// TIA Portal V17 export
// export: Created 2024-09-02T12:49:59.6784683Z, ExportSetting WithDefaults, DisplayName Totally Integrated Automation Portal, DisplayVersion V17, DisplayName TIA Portal Openness, DisplayVersion V17, DisplayName TIA Portal Version Control Interface, DisplayVersion V17, DisplayName STEP 7 Professional, DisplayVersion V17, DisplayName STEP 7 Safety, DisplayVersion V17, DisplayName WinCC Professional, DisplayVersion V17
FUNCTION_BLOCK "GraFB_Hand_21_30"   // FB1172, GRAPH
TITLE = GRAPH FB
AUTHOR : OlegFuehrus
FAMILY : SK
NAME : SK
VERSION : 0.1
// Hand functions / Handfunktionen
// stored: AcknowledgeErrorsRequired true, AutoNumber true, ExtensionBlockName LTLL_ManualGraphExt, GraphVersion 4.0, InitialValuesAcquisition false, IsIECCheckEnabled false, LanguageInNetworks LAD, LockOperatingMode false, PermanentILProcessingInMANMode true, SetENOAutomatically false, SkipSteps false, UDAEnableTagReadback false, WithAlarmHandling true
   // inherited from GRAPH_BASE
   VAR
      OFF_SQ_BASE : Bool;
   END_VAR
   VAR_INPUT
      OFF_SQ : Bool;
      INIT_SQ : Bool;
      ACK_EF : Bool;
      S_PREV : Bool;
      S_NEXT : Bool;
      SW_AUTO : Bool;
      SW_TAP : Bool;
      SW_MAN : Bool;
      S_SEL : Int;
      S_ON : Bool;
      S_OFF : Bool;
      T_PUSH : Bool;
   END_VAR
   VAR_OUTPUT
      S_NO : Int;
      S_MORE : Bool;
      S_ACTIVE : Bool;
      ERR_FLT : Bool;
      AUTO_ON : Bool;
      TAP_ON : Bool;
      MAN_ON : Bool;
   END_VAR
   VAR
      extBlock { S7_SetPoint := 'True'} : "LTLL_ManualGraphExt";
   END_VAR
   VAR_TEMP
      t_FrgHand : Bool;   // Freigabe Handbetrieb / Enable manual operation
      t_Service : Bool;   // Servicebetrieb aktiv / Service operation active
   END_VAR
BEGIN
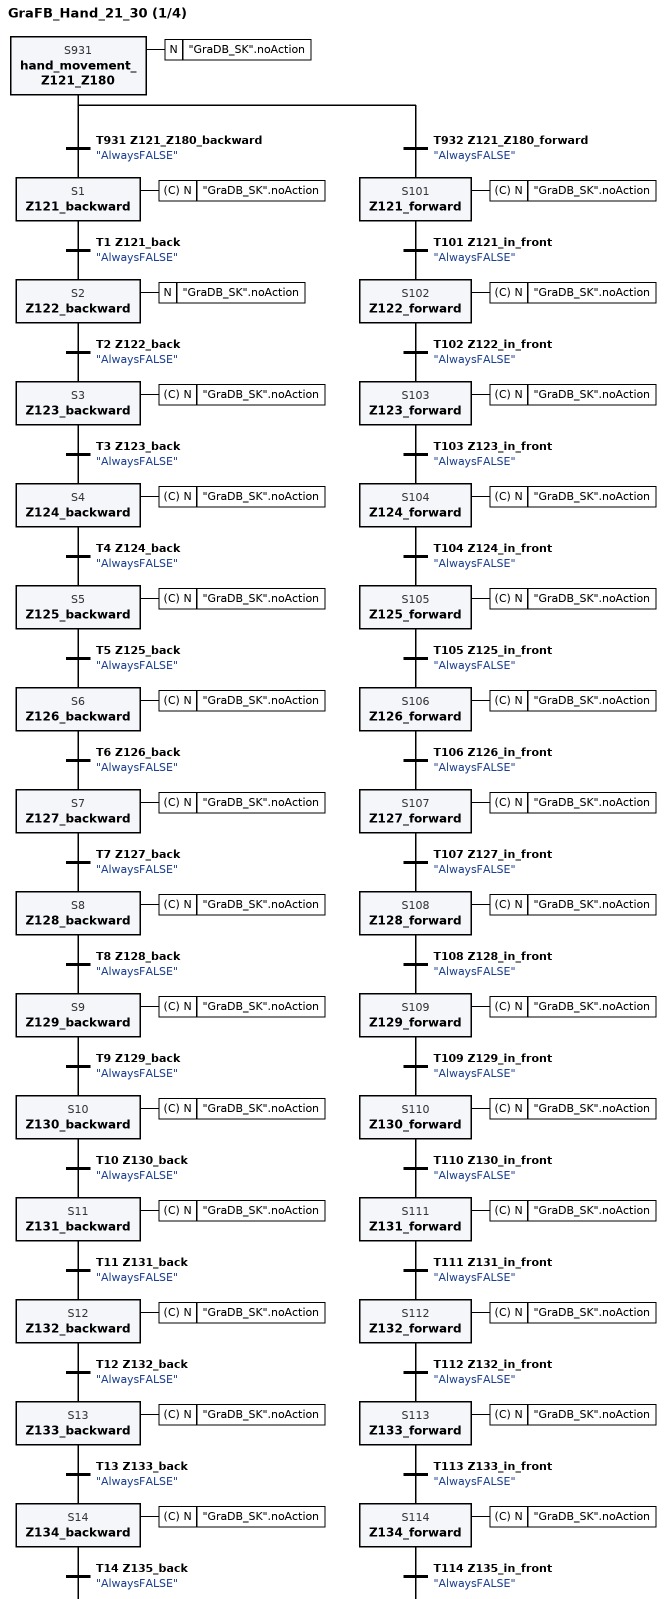
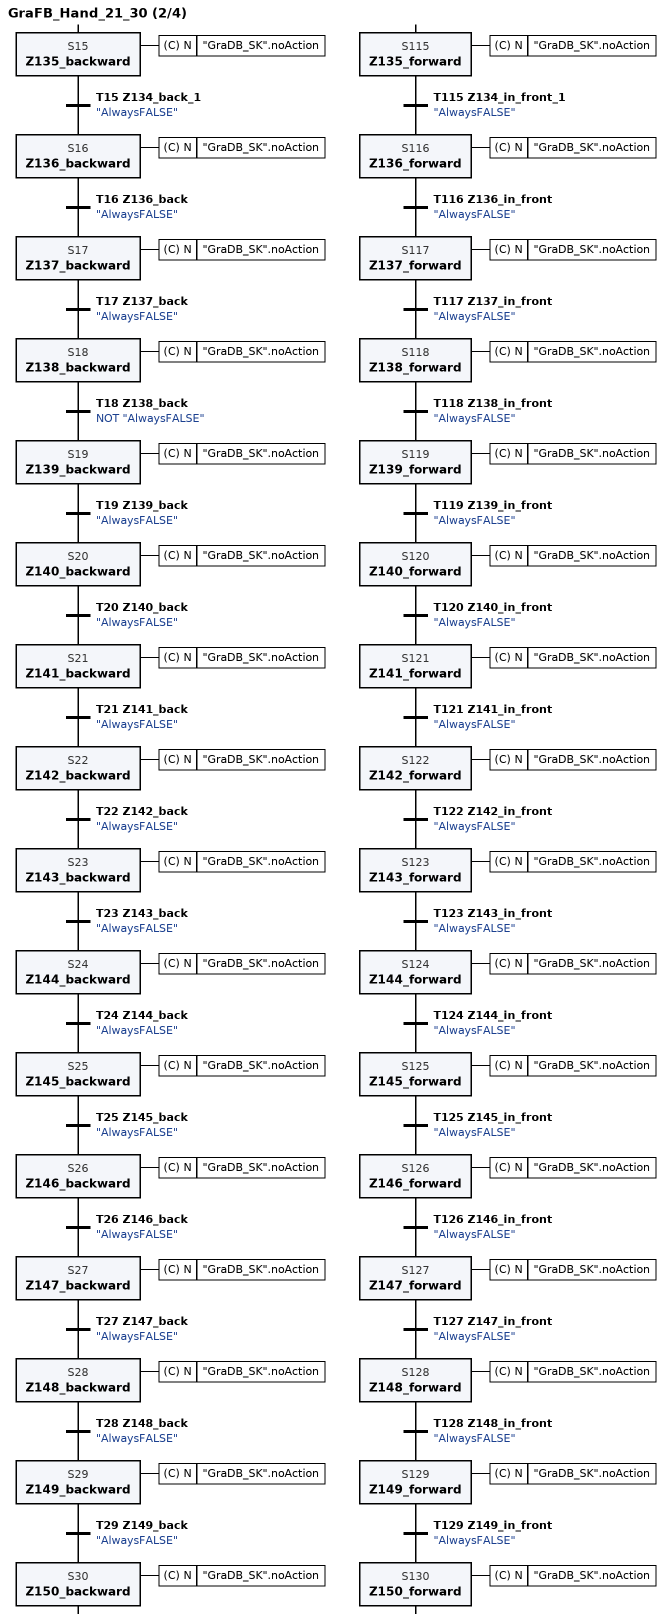
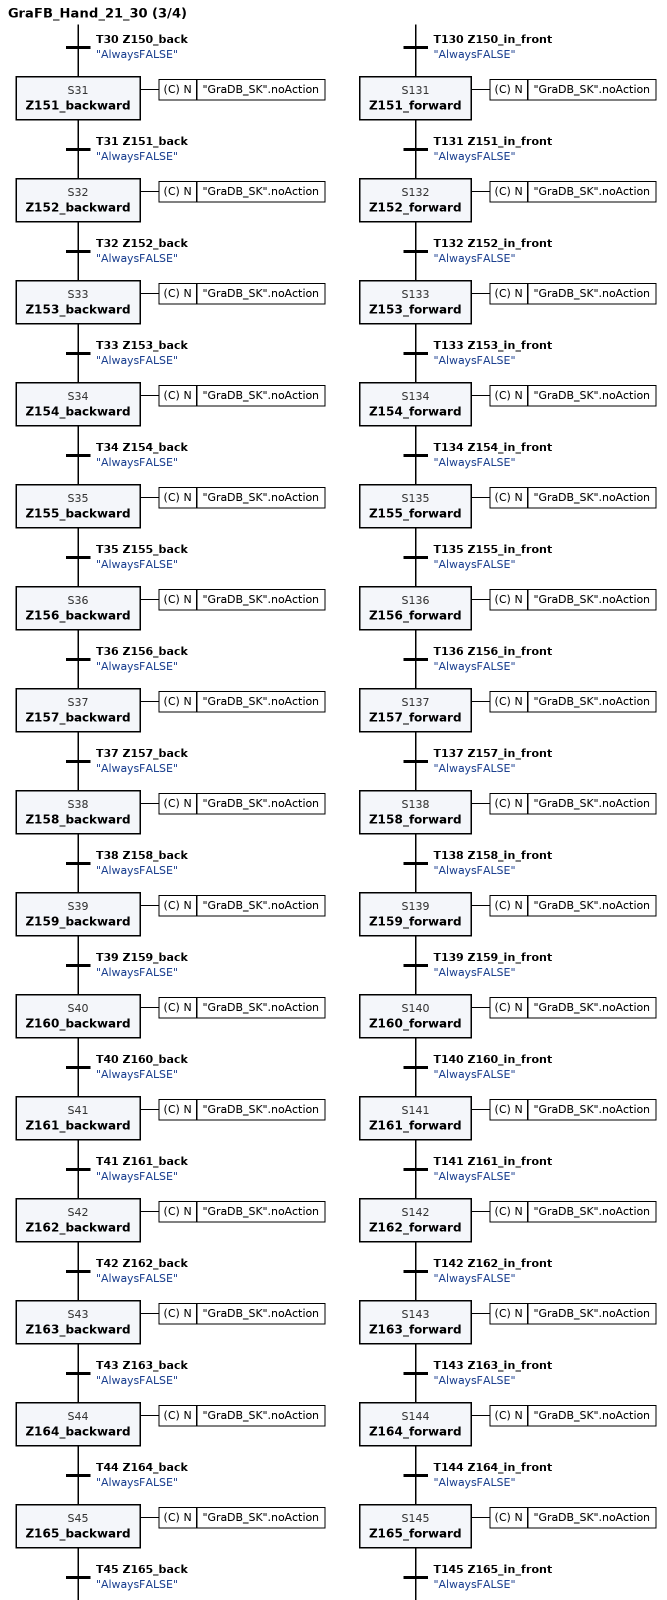
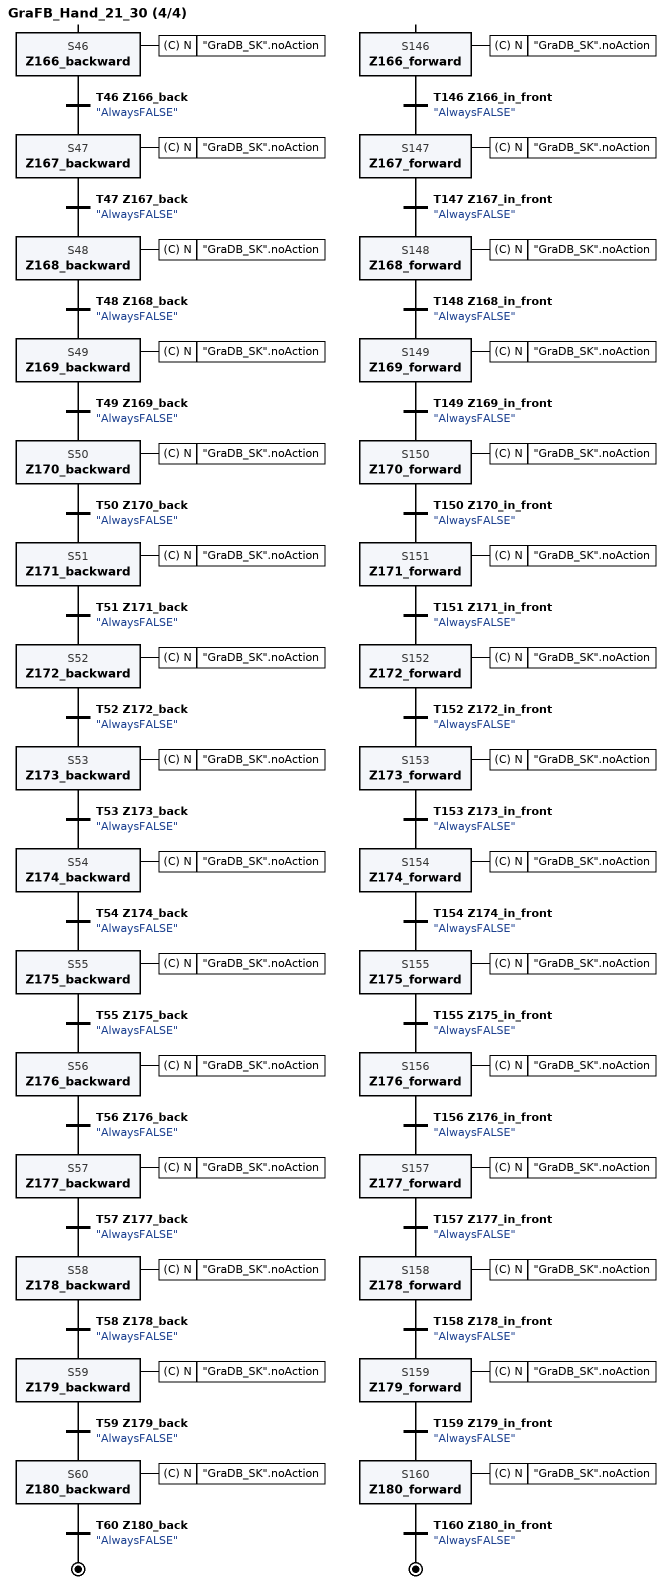
   // permanent pre-instructions
   NETWORK 1
   TITLE = HMI Lite Pass on data / HMI Lite Daten weiterreichen
      #extBlock.input := "LTLL_ManualGraphControl_OP70".screen[0].input;
   NETWORK 2
   TITLE = Instance DB Name query and pass on / Instanz DB Name abfragen und weiterreichen
      GetInstanceName(size := 0, OUT => #extBlock.input.instanceName);
   NETWORK 3
   TITLE = Interlocks Permanent machining, manual Approve and service / Interlocks Permanent Bearbeiten, Handfreigabe und Service
      IF NOT #RT_DATA.MOP.IL_PERM THEN #RT_DATA.MOP.IL_PERM := TRUE; END_IF;
      #t_FrgHand := "AnwDB_OperatingModes_OP70".BA[0]."mode_hand+start";
      #t_Service := "AnwDB_OperatingModes_OP70".BA[0].mode_service;

   // sequencer 1: Sequencer 1
   STEP hand_movement_Z121_Z180:   // S931, max time T#10S, warning time T#7S: Step commentary / Schrittkommentar
      interlock C := (none);   // hand_bereich_Z001_Z005
      supervision V := (none);   // hand_bereich_Z001_Z005
              N    "GraDB_SK".noAction
   END_STEP
   TRANSITION Z121_Z180_backward FROM hand_movement_Z121_Z180 TO Z121_backward   // T931
      := "AlwaysFALSE";
   END_TRANSITION
   TRANSITION Z121_Z180_forward FROM hand_movement_Z121_Z180 TO Z121_forward   // T932
      := "AlwaysFALSE";
   END_TRANSITION
   STEP Z121_backward:   // S1, max time T#10S, warning time T#7S
      interlock C := "AlwaysFALSE";   // Z121_zur
      supervision V := NOT #Z121_back.TT AND (#Z121_backward.T > T#5S);   // Z121_zur
      (C)     N    "GraDB_SK".noAction
   END_STEP
   TRANSITION Z121_back FROM Z121_backward TO Z122_backward   // T1
      := "AlwaysFALSE";
   END_TRANSITION
   STEP Z122_backward:   // S2, max time T#10S, warning time T#7S
      interlock C := "AlwaysFALSE";   // Z122_zur
      supervision V := NOT #Z122_back.TT AND (#Z122_backward.T > T#5S);   // Z122_zur
              N    "GraDB_SK".noAction
   END_STEP
   TRANSITION Z122_back FROM Z122_backward TO Z123_backward   // T2
      := "AlwaysFALSE";
   END_TRANSITION
   STEP Z123_backward:   // S3, max time T#10S, warning time T#7S
      interlock C := "AlwaysFALSE";   // Z123_zur
      supervision V := NOT #Z123_back.TT AND (#Z123_backward.T > T#5S);   // Z123_zur
      (C)     N    "GraDB_SK".noAction
   END_STEP
   TRANSITION Z123_back FROM Z123_backward TO Z124_backward   // T3
      := "AlwaysFALSE";
   END_TRANSITION
   STEP Z124_backward:   // S4, max time T#10S, warning time T#7S
      interlock C := "AlwaysFALSE";   // Z124_zur
      supervision V := NOT #Z124_back.TT AND (#Z124_backward.T > T#5S);   // Z124_zur
      (C)     N    "GraDB_SK".noAction
   END_STEP
   TRANSITION Z124_back FROM Z124_backward TO Z125_backward   // T4
      := "AlwaysFALSE";
   END_TRANSITION
   STEP Z125_backward:   // S5, max time T#10S, warning time T#7S
      interlock C := "AlwaysFALSE";   // Z125_zur
      supervision V := NOT #Z125_back.TT AND (#Z125_backward.T > T#5S);   // Z125_zur
      (C)     N    "GraDB_SK".noAction
   END_STEP
   TRANSITION Z125_back FROM Z125_backward TO Z126_backward   // T5
      := "AlwaysFALSE";
   END_TRANSITION
   STEP Z121_forward:   // S101, max time T#10S, warning time T#7S
      interlock C := "AlwaysFALSE";   // Z121_vor
      supervision V := NOT #Z121_in_front.TT AND (#Z121_forward.T > T#5S);   // Z121_vor
      (C)     N    "GraDB_SK".noAction
   END_STEP
   TRANSITION Z121_in_front FROM Z121_forward TO Z122_forward   // T101
      := "AlwaysFALSE";
   END_TRANSITION
   STEP Z122_forward:   // S102, max time T#10S, warning time T#7S
      interlock C := "AlwaysFALSE";   // Z122_vor
      supervision V := NOT #Z122_in_front.TT AND (#Z122_forward.T > T#5S);   // Z122_vor
      (C)     N    "GraDB_SK".noAction
   END_STEP
   TRANSITION Z122_in_front FROM Z122_forward TO Z123_forward   // T102
      := "AlwaysFALSE";
   END_TRANSITION
   STEP Z123_forward:   // S103, max time T#10S, warning time T#7S
      interlock C := "AlwaysFALSE";   // Z123_vor
      supervision V := NOT #Z123_in_front.TT AND (#Z123_forward.T > T#5S);   // Z123_vor
      (C)     N    "GraDB_SK".noAction
   END_STEP
   TRANSITION Z123_in_front FROM Z123_forward TO Z124_forward   // T103
      := "AlwaysFALSE";
   END_TRANSITION
   STEP Z124_forward:   // S104, max time T#10S, warning time T#7S
      interlock C := "AlwaysFALSE";   // Z124_vor
      supervision V := NOT #Z124_in_front.TT AND (#Z124_forward.T > T#5S);   // Z124_vor
      (C)     N    "GraDB_SK".noAction
   END_STEP
   TRANSITION Z124_in_front FROM Z124_forward TO Z125_forward   // T104
      := "AlwaysFALSE";
   END_TRANSITION
   STEP Z125_forward:   // S105, max time T#10S, warning time T#7S
      interlock C := "AlwaysFALSE";   // Z125_vor
      supervision V := NOT #Z125_in_front.TT AND (#Z125_forward.T > T#20S);   // Z125_vor
      (C)     N    "GraDB_SK".noAction
   END_STEP
   TRANSITION Z125_in_front FROM Z125_forward TO Z126_forward   // T105
      := "AlwaysFALSE";
   END_TRANSITION
   STEP Z126_backward:   // S6, max time T#10S, warning time T#7S: Cross transport 2 / Quertransport 2
      interlock C := "AlwaysFALSE";   // Z126_zur
      supervision V := NOT #Z126_back.TT AND (#Z126_backward.T > T#5S);   // Z126_zur
      (C)     N    "GraDB_SK".noAction
   END_STEP
   TRANSITION Z126_back FROM Z126_backward TO Z127_backward   // T6
      := "AlwaysFALSE";
   END_TRANSITION
   STEP Z127_backward:   // S7, max time T#10S, warning time T#7S
      interlock C := "AlwaysFALSE";   // Z127_zur
      supervision V := NOT #Z127_back.TT AND (#Z127_backward.T > T#5S);   // Z127_zur
      (C)     N    "GraDB_SK".noAction
   END_STEP
   TRANSITION Z127_back FROM Z127_backward TO Z128_backward   // T7
      := "AlwaysFALSE";
   END_TRANSITION
   STEP Z128_backward:   // S8, max time T#10S, warning time T#7S
      interlock C := "AlwaysFALSE";   // Z128_zur
      supervision V := NOT #Z128_back.TT AND (#Z128_backward.T > T#5S);   // Z128_zur
      (C)     N    "GraDB_SK".noAction
   END_STEP
   TRANSITION Z128_back FROM Z128_backward TO Z129_backward   // T8
      := "AlwaysFALSE";
   END_TRANSITION
   STEP Z129_backward:   // S9, max time T#10S, warning time T#7S
      interlock C := "AlwaysFALSE";   // Z129_zur
      supervision V := NOT #Z129_back.TT AND (#Z129_backward.T > T#5S);   // Z129_zur
      (C)     N    "GraDB_SK".noAction
   END_STEP
   TRANSITION Z129_back FROM Z129_backward TO Z130_backward   // T9
      := "AlwaysFALSE";
   END_TRANSITION
   STEP Z130_backward:   // S10, max time T#10S, warning time T#7S
      interlock C := "AlwaysFALSE";   // Z130_zur
      supervision V := NOT #Z130_back.TT AND (#Z130_backward.T > T#5S);   // Z130_zur
      (C)     N    "GraDB_SK".noAction
   END_STEP
   TRANSITION Z130_back FROM Z130_backward TO Z131_backward   // T10
      := "AlwaysFALSE";
   END_TRANSITION
   STEP Z126_forward:   // S106, max time T#10S, warning time T#7S
      interlock C := "AlwaysFALSE";   // Z126_vor
      supervision V := NOT #Z126_in_front.TT AND (#Z126_forward.T > T#5S);   // Z126_vor
      (C)     N    "GraDB_SK".noAction
   END_STEP
   TRANSITION Z126_in_front FROM Z126_forward TO Z127_forward   // T106
      := "AlwaysFALSE";
   END_TRANSITION
   STEP Z127_forward:   // S107, max time T#10S, warning time T#7S
      interlock C := "AlwaysFALSE";   // Z127_vor
      supervision V := NOT #Z127_in_front.TT AND (#Z127_forward.T > T#5S);   // Z127_vor
      (C)     N    "GraDB_SK".noAction
   END_STEP
   TRANSITION Z127_in_front FROM Z127_forward TO Z128_forward   // T107
      := "AlwaysFALSE";
   END_TRANSITION
   STEP Z128_forward:   // S108, max time T#10S, warning time T#7S
      interlock C := "AlwaysFALSE";   // Z128_vor
      supervision V := NOT #Z128_in_front.TT AND (#Z128_forward.T > T#5S);   // Z128_vor
      (C)     N    "GraDB_SK".noAction
   END_STEP
   TRANSITION Z128_in_front FROM Z128_forward TO Z129_forward   // T108
      := "AlwaysFALSE";
   END_TRANSITION
   STEP Z129_forward:   // S109, max time T#10S, warning time T#7S
      interlock C := "AlwaysFALSE";   // Z129_vor
      supervision V := NOT #Z129_in_front.TT AND (#Z129_forward.T > T#5S);   // Z129_vor
      (C)     N    "GraDB_SK".noAction
   END_STEP
   TRANSITION Z129_in_front FROM Z129_forward TO Z130_forward   // T109
      := "AlwaysFALSE";
   END_TRANSITION
   STEP Z130_forward:   // S110, max time T#10S, warning time T#7S
      interlock C := "AlwaysFALSE";   // Z130_vor
      supervision V := NOT #Z130_in_front.TT AND (#Z130_forward.T > T#5S);   // Z130_vor
      (C)     N    "GraDB_SK".noAction
   END_STEP
   TRANSITION Z130_in_front FROM Z130_forward TO Z131_forward   // T110
      := "AlwaysFALSE";
   END_TRANSITION
   STEP Z131_backward:   // S11, max time T#10S, warning time T#7S
      interlock C := "AlwaysFALSE";   // Z131_zur
      supervision V := NOT #Z131_back.TT AND (#Z131_backward.T > T#5S);   // Z131_zur
      (C)     N    "GraDB_SK".noAction
   END_STEP
   TRANSITION Z131_back FROM Z131_backward TO Z132_backward   // T11
      := "AlwaysFALSE";
   END_TRANSITION
   STEP Z132_backward:   // S12, max time T#10S, warning time T#7S
      interlock C := "AlwaysFALSE";   // Z132_zur
      supervision V := NOT #Z132_back.TT AND (#Z132_backward.T > T#5S);   // Z132_zur
      (C)     N    "GraDB_SK".noAction
   END_STEP
   TRANSITION Z132_back FROM Z132_backward TO Z133_backward   // T12
      := "AlwaysFALSE";
   END_TRANSITION
   STEP Z133_backward:   // S13, max time T#10S, warning time T#7S
      interlock C := "AlwaysFALSE";   // Z133_zur
      supervision V := NOT #Z133_back.TT AND (#Z133_backward.T > T#5S);   // Z133_zur
      (C)     N    "GraDB_SK".noAction
   END_STEP
   TRANSITION Z133_back FROM Z133_backward TO Z134_backward   // T13
      := "AlwaysFALSE";
   END_TRANSITION
   STEP Z134_backward:   // S14, max time T#10S, warning time T#7S
      interlock C := "AlwaysFALSE";   // Z135_zur
      supervision V := NOT #Z135_back.TT AND (#Z134_backward.T > T#5S);   // Z135_zur
      (C)     N    "GraDB_SK".noAction
   END_STEP
   TRANSITION Z135_back FROM Z134_backward TO Z135_backward   // T14
      := "AlwaysFALSE";
   END_TRANSITION
   STEP Z135_backward:   // S15, max time T#10S, warning time T#7S
      interlock C := "AlwaysFALSE";   // Z134_zur
      supervision V := NOT #Z136_back.TT AND (#Z135_backward.T > T#5S);   // Z134_zur
      (C)     N    "GraDB_SK".noAction
   END_STEP
   TRANSITION Z134_back_1 FROM Z135_backward TO Z136_backward   // T15
      := "AlwaysFALSE";
   END_TRANSITION
   STEP Z131_forward:   // S111, max time T#10S, warning time T#7S
      interlock C := "AlwaysFALSE";   // Z131_vor
      supervision V := NOT #Z131_in_front.TT AND (#Z131_forward.T > T#5S);   // Z131_vor
      (C)     N    "GraDB_SK".noAction
   END_STEP
   TRANSITION Z131_in_front FROM Z131_forward TO Z132_forward   // T111
      := "AlwaysFALSE";
   END_TRANSITION
   STEP Z132_forward:   // S112, max time T#10S, warning time T#7S
      interlock C := "AlwaysFALSE";   // Z132_vor
      supervision V := NOT #Z132_in_front.TT AND (#Z132_forward.T > T#5S);   // Z132_vor
      (C)     N    "GraDB_SK".noAction
   END_STEP
   TRANSITION Z132_in_front FROM Z132_forward TO Z133_forward   // T112
      := "AlwaysFALSE";
   END_TRANSITION
   STEP Z133_forward:   // S113, max time T#10S, warning time T#7S
      interlock C := "AlwaysFALSE";   // Z133_vor
      supervision V := NOT #Z133_in_front.TT AND (#Z133_forward.T > T#5S);   // Z133_vor
      (C)     N    "GraDB_SK".noAction
   END_STEP
   TRANSITION Z133_in_front FROM Z133_forward TO Z134_forward   // T113
      := "AlwaysFALSE";
   END_TRANSITION
   STEP Z134_forward:   // S114, max time T#10S, warning time T#7S
      interlock C := "AlwaysFALSE";   // Z135_vor
      supervision V := NOT #Z135_in_front.TT AND (#Z134_forward.T > T#5S);   // Z135_vor
      (C)     N    "GraDB_SK".noAction
   END_STEP
   TRANSITION Z135_in_front FROM Z134_forward TO Z135_forward   // T114
      := "AlwaysFALSE";
   END_TRANSITION
   STEP Z135_forward:   // S115, max time T#10S, warning time T#7S
      interlock C := "AlwaysFALSE";   // Z134_vor
      supervision V := NOT #Z136_in_front.TT AND (#Z135_forward.T > T#5S);   // Z134_vor
      (C)     N    "GraDB_SK".noAction
   END_STEP
   TRANSITION Z134_in_front_1 FROM Z135_forward TO Z136_forward   // T115
      := "AlwaysFALSE";
   END_TRANSITION
   STEP Z136_backward:   // S16, max time T#10S, warning time T#7S
      interlock C := "AlwaysFALSE";   // Z136_zur
      supervision V := NOT #Z136_back.TT AND (#Z136_backward.T > T#5S);   // Z136_zur
      (C)     N    "GraDB_SK".noAction
   END_STEP
   TRANSITION Z136_back FROM Z136_backward TO Z137_backward   // T16
      := "AlwaysFALSE";
   END_TRANSITION
   STEP Z137_backward:   // S17, max time T#10S, warning time T#7S
      interlock C := "AlwaysFALSE";   // Z137_zur
      supervision V := NOT #Z137_back.TT AND (#Z137_backward.T > T#5S);   // Z137_zur
      (C)     N    "GraDB_SK".noAction
   END_STEP
   TRANSITION Z137_back FROM Z137_backward TO Z138_backward   // T17
      := "AlwaysFALSE";
   END_TRANSITION
   STEP Z138_backward:   // S18, max time T#10S, warning time T#7S
      interlock C := "AlwaysFALSE";   // Z138_zur
      supervision V := NOT #Z138_back.TT AND (#Z138_backward.T > T#5S);   // Z138_zur
      (C)     N    "GraDB_SK".noAction
   END_STEP
   TRANSITION Z138_back FROM Z138_backward TO Z139_backward   // T18
      := NOT "AlwaysFALSE";
   END_TRANSITION
   STEP Z139_backward:   // S19, max time T#10S, warning time T#7S
      interlock C := "AlwaysFALSE";   // Z139_zur
      supervision V := NOT #Z139_back.TT AND (#Z139_backward.T > T#5S);   // Z139_zur
      (C)     N    "GraDB_SK".noAction
   END_STEP
   TRANSITION Z139_back FROM Z139_backward TO Z140_backward   // T19
      := "AlwaysFALSE";
   END_TRANSITION
   STEP Z140_backward:   // S20, max time T#10S, warning time T#7S
      interlock C := "AlwaysFALSE";   // Z140_zur
      supervision V := NOT #Z140_back.TT AND (#Z140_backward.T > T#5S);   // Z140_zur
      (C)     N    "GraDB_SK".noAction
   END_STEP
   TRANSITION Z140_back FROM Z140_backward TO Z141_backward   // T20
      := "AlwaysFALSE";
   END_TRANSITION
   STEP Z136_forward:   // S116, max time T#10S, warning time T#7S
      interlock C := "AlwaysFALSE";   // Z136_vor
      supervision V := NOT #Z136_in_front.TT AND (#Z136_forward.T > T#5S);   // Z136_vor
      (C)     N    "GraDB_SK".noAction
   END_STEP
   TRANSITION Z136_in_front FROM Z136_forward TO Z137_forward   // T116
      := "AlwaysFALSE";
   END_TRANSITION
   STEP Z137_forward:   // S117, max time T#10S, warning time T#7S
      interlock C := "AlwaysFALSE";   // Z137_vor
      supervision V := NOT #Z137_in_front.TT AND (#Z137_forward.T > T#5S);   // Z137_vor
      (C)     N    "GraDB_SK".noAction
   END_STEP
   TRANSITION Z137_in_front FROM Z137_forward TO Z138_forward   // T117
      := "AlwaysFALSE";
   END_TRANSITION
   STEP Z138_forward:   // S118, max time T#10S, warning time T#7S
      interlock C := "AlwaysFALSE";   // Z138_vor
      supervision V := NOT #Z138_in_front.TT AND (#Z138_forward.T > T#5S);   // Z138_vor
      (C)     N    "GraDB_SK".noAction
   END_STEP
   TRANSITION Z138_in_front FROM Z138_forward TO Z139_forward   // T118
      := "AlwaysFALSE";
   END_TRANSITION
   STEP Z139_forward:   // S119, max time T#10S, warning time T#7S
      interlock C := "AlwaysFALSE";   // Z139_vor
      supervision V := NOT #Z139_in_front.TT AND (#Z139_forward.T > T#5S);   // Z139_vor
      (C)     N    "GraDB_SK".noAction
   END_STEP
   TRANSITION Z139_in_front FROM Z139_forward TO Z140_forward   // T119
      := "AlwaysFALSE";
   END_TRANSITION
   STEP Z140_forward:   // S120, max time T#10S, warning time T#7S
      interlock C := "AlwaysFALSE";   // Z140_vor
      supervision V := NOT #Z140_in_front.TT AND (#Z140_forward.T > T#5S);   // Z140_vor
      (C)     N    "GraDB_SK".noAction
   END_STEP
   TRANSITION Z140_in_front FROM Z140_forward TO Z141_forward   // T120
      := "AlwaysFALSE";
   END_TRANSITION
   STEP Z141_backward:   // S21, max time T#10S, warning time T#7S
      interlock C := "AlwaysFALSE";   // Z141_zur
      supervision V := NOT #Z141_back.TT AND (#Z141_backward.T > T#10S);   // Z141_zur
      (C)     N    "GraDB_SK".noAction
   END_STEP
   TRANSITION Z141_back FROM Z141_backward TO Z142_backward   // T21
      := "AlwaysFALSE";
   END_TRANSITION
   STEP Z142_backward:   // S22, max time T#10S, warning time T#7S
      interlock C := "AlwaysFALSE";   // Z142_zur
      supervision V := NOT #Z142_back.TT AND (#Z142_backward.T > T#10S);   // Z142_zur
      (C)     N    "GraDB_SK".noAction
   END_STEP
   TRANSITION Z142_back FROM Z142_backward TO Z143_backward   // T22
      := "AlwaysFALSE";
   END_TRANSITION
   STEP Z143_backward:   // S23, max time T#10S, warning time T#7S
      interlock C := "AlwaysFALSE";   // Z143_zur
      supervision V := NOT #Z143_back.TT AND (#Z143_backward.T > T#10S);   // Z143_zur
      (C)     N    "GraDB_SK".noAction
   END_STEP
   TRANSITION Z143_back FROM Z143_backward TO Z144_backward   // T23
      := "AlwaysFALSE";
   END_TRANSITION
   STEP Z144_backward:   // S24, max time T#10S, warning time T#7S
      interlock C := "AlwaysFALSE";   // Z144_zur
      supervision V := NOT #Z144_back.TT AND (#Z144_backward.T > T#5S);   // Z144_zur
      (C)     N    "GraDB_SK".noAction
   END_STEP
   TRANSITION Z144_back FROM Z144_backward TO Z145_backward   // T24
      := "AlwaysFALSE";
   END_TRANSITION
   STEP Z145_backward:   // S25, max time T#10S, warning time T#7S
      interlock C := "AlwaysFALSE";   // Z145_zur
      supervision V := NOT #Z145_back.TT AND (#Z145_backward.T > T#5S);   // Z145_zur
      (C)     N    "GraDB_SK".noAction
   END_STEP
   TRANSITION Z145_back FROM Z145_backward TO Z146_backward   // T25
      := "AlwaysFALSE";
   END_TRANSITION
   STEP Z141_forward:   // S121, max time T#10S, warning time T#7S
      interlock C := "AlwaysFALSE";   // Z141_vor
      supervision V := NOT #Z141_in_front.TT AND (#Z141_forward.T > T#5S);   // Z141_vor
      (C)     N    "GraDB_SK".noAction
   END_STEP
   TRANSITION Z141_in_front FROM Z141_forward TO Z142_forward   // T121
      := "AlwaysFALSE";
   END_TRANSITION
   STEP Z142_forward:   // S122, max time T#10S, warning time T#7S
      interlock C := "AlwaysFALSE";   // Z142_vor
      supervision V := NOT #Z142_in_front.TT AND (#Z142_forward.T > T#10S);   // Z142_vor
      (C)     N    "GraDB_SK".noAction
   END_STEP
   TRANSITION Z142_in_front FROM Z142_forward TO Z143_forward   // T122
      := "AlwaysFALSE";
   END_TRANSITION
   STEP Z143_forward:   // S123, max time T#10S, warning time T#7S
      interlock C := "AlwaysFALSE";   // Z143_vor
      supervision V := NOT #Z143_in_front.TT AND (#Z143_forward.T > T#10S);   // Z143_vor
      (C)     N    "GraDB_SK".noAction
   END_STEP
   TRANSITION Z143_in_front FROM Z143_forward TO Z144_forward   // T123
      := "AlwaysFALSE";
   END_TRANSITION
   STEP Z144_forward:   // S124, max time T#10S, warning time T#7S
      interlock C := "AlwaysFALSE";   // Z144_vor
      supervision V := NOT #Z144_in_front.TT AND (#Z144_forward.T > T#5S);   // Z144_vor
      (C)     N    "GraDB_SK".noAction
   END_STEP
   TRANSITION Z144_in_front FROM Z144_forward TO Z145_forward   // T124
      := "AlwaysFALSE";
   END_TRANSITION
   STEP Z145_forward:   // S125, max time T#10S, warning time T#7S
      interlock C := "AlwaysFALSE";   // Z145_vor
      supervision V := NOT #Z145_in_front.TT AND (#Z145_forward.T > T#5S);   // Z145_vor
      (C)     N    "GraDB_SK".noAction
   END_STEP
   TRANSITION Z145_in_front FROM Z145_forward TO Z146_forward   // T125
      := "AlwaysFALSE";
   END_TRANSITION
   STEP Z146_backward:   // S26, max time T#10S, warning time T#7S
      interlock C := "AlwaysFALSE";   // Z146_zur
      supervision V := NOT #Z146_back.TT AND (#Z146_backward.T > T#5S);   // Z146_zur
      (C)     N    "GraDB_SK".noAction
   END_STEP
   TRANSITION Z146_back FROM Z146_backward TO Z147_backward   // T26
      := "AlwaysFALSE";
   END_TRANSITION
   STEP Z147_backward:   // S27, max time T#10S, warning time T#7S
      interlock C := "AlwaysFALSE";   // Z147_zur
      supervision V := NOT #Z147_back.TT AND (#Z147_backward.T > T#5S);   // Z147_zur
      (C)     N    "GraDB_SK".noAction
   END_STEP
   TRANSITION Z147_back FROM Z147_backward TO Z148_backward   // T27
      := "AlwaysFALSE";
   END_TRANSITION
   STEP Z148_backward:   // S28, max time T#10S, warning time T#7S
      interlock C := "AlwaysFALSE";   // Z148_zur
      supervision V := NOT #Z148_back.TT AND (#Z148_backward.T > T#5S);   // Z148_zur
      (C)     N    "GraDB_SK".noAction
   END_STEP
   TRANSITION Z148_back FROM Z148_backward TO Z149_backward   // T28
      := "AlwaysFALSE";
   END_TRANSITION
   STEP Z149_backward:   // S29, max time T#10S, warning time T#7S
      interlock C := "AlwaysFALSE";   // Z149_zur
      supervision V := NOT #Z149_back.TT AND (#Z149_backward.T > T#5S);   // Z149_zur
      (C)     N    "GraDB_SK".noAction
   END_STEP
   TRANSITION Z149_back FROM Z149_backward TO Z150_backward   // T29
      := "AlwaysFALSE";
   END_TRANSITION
   STEP Z150_backward:   // S30, max time T#10S, warning time T#7S
      interlock C := "AlwaysFALSE";   // Z150_zur
      supervision V := NOT #Z150_back.TT AND (#Z150_backward.T > T#5S);   // Z150_zur
      (C)     N    "GraDB_SK".noAction
   END_STEP
   TRANSITION Z150_back FROM Z150_backward TO Z151_backward   // T30
      := "AlwaysFALSE";
   END_TRANSITION
   STEP Z146_forward:   // S126, max time T#10S, warning time T#7S
      interlock C := "AlwaysFALSE";   // Z146_vor
      supervision V := NOT #Z146_in_front.TT AND (#Z146_forward.T > T#5S);   // Z146_vor
      (C)     N    "GraDB_SK".noAction
   END_STEP
   TRANSITION Z146_in_front FROM Z146_forward TO Z147_forward   // T126
      := "AlwaysFALSE";
   END_TRANSITION
   STEP Z147_forward:   // S127, max time T#10S, warning time T#7S
      interlock C := "AlwaysFALSE";   // Z147_vor
      supervision V := NOT #Z147_in_front.TT AND (#Z147_forward.T > T#5S);   // Z147_vor
      (C)     N    "GraDB_SK".noAction
   END_STEP
   TRANSITION Z147_in_front FROM Z147_forward TO Z148_forward   // T127
      := "AlwaysFALSE";
   END_TRANSITION
   STEP Z148_forward:   // S128, max time T#10S, warning time T#7S
      interlock C := "AlwaysFALSE";   // Z148_vor
      supervision V := NOT #Z148_in_front.TT AND (#Z148_forward.T > T#5S);   // Z148_vor
      (C)     N    "GraDB_SK".noAction
   END_STEP
   TRANSITION Z148_in_front FROM Z148_forward TO Z149_forward   // T128
      := "AlwaysFALSE";
   END_TRANSITION
   STEP Z149_forward:   // S129, max time T#10S, warning time T#7S
      interlock C := "AlwaysFALSE";   // Z149_vor
      supervision V := NOT #Z149_in_front.TT AND (#Z149_forward.T > T#5S);   // Z149_vor
      (C)     N    "GraDB_SK".noAction
   END_STEP
   TRANSITION Z149_in_front FROM Z149_forward TO Z150_forward   // T129
      := "AlwaysFALSE";
   END_TRANSITION
   STEP Z150_forward:   // S130, max time T#10S, warning time T#7S
      interlock C := "AlwaysFALSE";   // Z150_vor
      supervision V := NOT #Z150_in_front.TT AND (#Z150_forward.T > T#5S);   // Z150_vor
      (C)     N    "GraDB_SK".noAction
   END_STEP
   TRANSITION Z150_in_front FROM Z150_forward TO Z151_forward   // T130
      := "AlwaysFALSE";
   END_TRANSITION
   STEP Z151_backward:   // S31, max time T#10S, warning time T#7S: Step commentary / Schrittkommentar
      interlock C := "AlwaysFALSE";   // Z151_zur
      supervision V := NOT #Z151_back.TT AND (#Z151_backward.T > T#5S);   // Z151_zur
      (C)     N    "GraDB_SK".noAction
   END_STEP
   TRANSITION Z151_back FROM Z151_backward TO Z152_backward   // T31
      := "AlwaysFALSE";
   END_TRANSITION
   STEP Z152_backward:   // S32, max time T#10S, warning time T#7S: Step commentary / Schrittkommentar
      interlock C := "AlwaysFALSE";   // Z152_zur
      supervision V := NOT #Z152_back.TT AND (#Z152_backward.T > T#5S);   // Z152_zur
      (C)     N    "GraDB_SK".noAction
   END_STEP
   TRANSITION Z152_back FROM Z152_backward TO Z153_backward   // T32
      := "AlwaysFALSE";
   END_TRANSITION
   STEP Z153_backward:   // S33, max time T#10S, warning time T#7S: Step commentary / Schrittkommentar
      interlock C := "AlwaysFALSE";   // Z153_zur
      supervision V := NOT #Z153_back.TT AND (#Z153_backward.T > T#5S);   // Z153_zur
      (C)     N    "GraDB_SK".noAction
   END_STEP
   TRANSITION Z153_back FROM Z153_backward TO Z154_backward   // T33
      := "AlwaysFALSE";
   END_TRANSITION
   STEP Z154_backward:   // S34, max time T#10S, warning time T#7S: Step commentary / Schrittkommentar
      interlock C := "AlwaysFALSE";   // Z154_zur
      supervision V := NOT #Z154_back.TT AND (#Z154_backward.T > T#5S);   // Z154_zur
      (C)     N    "GraDB_SK".noAction
   END_STEP
   TRANSITION Z154_back FROM Z154_backward TO Z155_backward   // T34
      := "AlwaysFALSE";
   END_TRANSITION
   STEP Z155_backward:   // S35, max time T#10S, warning time T#7S: Step commentary / Schrittkommentar
      interlock C := "AlwaysFALSE";   // Z155_zur
      supervision V := NOT #Z155_back.TT AND (#Z155_backward.T > T#5S);   // Z155_zur
      (C)     N    "GraDB_SK".noAction
   END_STEP
   TRANSITION Z155_back FROM Z155_backward TO Z156_backward   // T35
      := "AlwaysFALSE";
   END_TRANSITION
   STEP Z151_forward:   // S131, max time T#10S, warning time T#7S: Step commentary / Schrittkommentar
      interlock C := "AlwaysFALSE";   // Z151_vor
      supervision V := NOT #Z151_in_front.TT AND (#Z151_forward.T > T#5S);   // Z151_vor
      (C)     N    "GraDB_SK".noAction
   END_STEP
   TRANSITION Z151_in_front FROM Z151_forward TO Z152_forward   // T131
      := "AlwaysFALSE";
   END_TRANSITION
   STEP Z152_forward:   // S132, max time T#10S, warning time T#7S: Step commentary / Schrittkommentar
      interlock C := "AlwaysFALSE";   // Z152_vor
      supervision V := NOT #Z152_in_front.TT AND (#Z152_forward.T > T#5S);   // Z152_vor
      (C)     N    "GraDB_SK".noAction
   END_STEP
   TRANSITION Z152_in_front FROM Z152_forward TO Z153_forward   // T132
      := "AlwaysFALSE";
   END_TRANSITION
   STEP Z153_forward:   // S133, max time T#10S, warning time T#7S: Step commentary / Schrittkommentar
      interlock C := "AlwaysFALSE";   // Z153_vor
      supervision V := NOT #Z153_in_front.TT AND (#Z153_forward.T > T#5S);   // Z153_vor
      (C)     N    "GraDB_SK".noAction
   END_STEP
   TRANSITION Z153_in_front FROM Z153_forward TO Z154_forward   // T133
      := "AlwaysFALSE";
   END_TRANSITION
   STEP Z154_forward:   // S134, max time T#10S, warning time T#7S: Step commentary / Schrittkommentar
      interlock C := "AlwaysFALSE";   // Z154_vor
      supervision V := NOT #Z154_in_front.TT AND (#Z154_forward.T > T#5S);   // Z154_vor
      (C)     N    "GraDB_SK".noAction
   END_STEP
   TRANSITION Z154_in_front FROM Z154_forward TO Z155_forward   // T134
      := "AlwaysFALSE";
   END_TRANSITION
   STEP Z155_forward:   // S135, max time T#10S, warning time T#7S: Step commentary / Schrittkommentar
      interlock C := "AlwaysFALSE";   // Z155_vor
      supervision V := NOT #Z155_in_front.TT AND (#Z155_forward.T > T#5S);   // Z155_vor
      (C)     N    "GraDB_SK".noAction
   END_STEP
   TRANSITION Z155_in_front FROM Z155_forward TO Z156_forward   // T135
      := "AlwaysFALSE";
   END_TRANSITION
   STEP Z156_backward:   // S36, max time T#10S, warning time T#7S: Step commentary / Schrittkommentar
      interlock C := "AlwaysFALSE";   // Z156_zur
      supervision V := NOT #Z156_back.TT AND (#Z156_backward.T > T#5S);   // Z156_zur
      (C)     N    "GraDB_SK".noAction
   END_STEP
   TRANSITION Z156_back FROM Z156_backward TO Z157_backward   // T36
      := "AlwaysFALSE";
   END_TRANSITION
   STEP Z157_backward:   // S37, max time T#10S, warning time T#7S: Step commentary / Schrittkommentar
      interlock C := "AlwaysFALSE";   // Z157_zur
      supervision V := NOT #Z157_back.TT AND (#Z157_backward.T > T#5S);   // Z157_zur
      (C)     N    "GraDB_SK".noAction
   END_STEP
   TRANSITION Z157_back FROM Z157_backward TO Z158_backward   // T37
      := "AlwaysFALSE";
   END_TRANSITION
   STEP Z158_backward:   // S38, max time T#10S, warning time T#7S: Step commentary / Schrittkommentar
      interlock C := "AlwaysFALSE";   // Z158_zur
      supervision V := NOT #Z158_back.TT AND (#Z158_backward.T > T#5S);   // Z158_zur
      (C)     N    "GraDB_SK".noAction
   END_STEP
   TRANSITION Z158_back FROM Z158_backward TO Z159_backward   // T38
      := "AlwaysFALSE";
   END_TRANSITION
   STEP Z159_backward:   // S39, max time T#10S, warning time T#7S: Step commentary / Schrittkommentar
      interlock C := "AlwaysFALSE";   // Z159_zur
      supervision V := NOT #Z159_back.TT AND (#Z159_backward.T > T#5S);   // Z159_zur
      (C)     N    "GraDB_SK".noAction
   END_STEP
   TRANSITION Z159_back FROM Z159_backward TO Z160_backward   // T39
      := "AlwaysFALSE";
   END_TRANSITION
   STEP Z160_backward:   // S40, max time T#10S, warning time T#7S: Step commentary / Schrittkommentar
      interlock C := "AlwaysFALSE";   // Z160_zur
      supervision V := NOT #Z160_back.TT AND (#Z160_backward.T > T#5S);   // Z160_zur
      (C)     N    "GraDB_SK".noAction
   END_STEP
   TRANSITION Z160_back FROM Z160_backward TO Z161_backward   // T40
      := "AlwaysFALSE";
   END_TRANSITION
   STEP Z156_forward:   // S136, max time T#10S, warning time T#7S: Step commentary / Schrittkommentar
      interlock C := "AlwaysFALSE";   // Z156_vor
      supervision V := NOT #Z156_in_front.TT AND (#Z156_forward.T > T#5S);   // Z156_vor
      (C)     N    "GraDB_SK".noAction
   END_STEP
   TRANSITION Z156_in_front FROM Z156_forward TO Z157_forward   // T136
      := "AlwaysFALSE";
   END_TRANSITION
   STEP Z157_forward:   // S137, max time T#10S, warning time T#7S: Step commentary / Schrittkommentar
      interlock C := "AlwaysFALSE";   // Z157_vor
      supervision V := NOT #Z157_in_front.TT AND (#Z157_forward.T > T#5S);   // Z157_vor
      (C)     N    "GraDB_SK".noAction
   END_STEP
   TRANSITION Z157_in_front FROM Z157_forward TO Z158_forward   // T137
      := "AlwaysFALSE";
   END_TRANSITION
   STEP Z158_forward:   // S138, max time T#10S, warning time T#7S: Step commentary / Schrittkommentar
      interlock C := "AlwaysFALSE";   // Z158_vor
      supervision V := NOT #Z158_in_front.TT AND (#Z158_forward.T > T#5S);   // Z158_vor
      (C)     N    "GraDB_SK".noAction
   END_STEP
   TRANSITION Z158_in_front FROM Z158_forward TO Z159_forward   // T138
      := "AlwaysFALSE";
   END_TRANSITION
   STEP Z159_forward:   // S139, max time T#10S, warning time T#7S: Step commentary / Schrittkommentar
      interlock C := "AlwaysFALSE";   // Z159_vor
      supervision V := NOT #Z159_in_front.TT AND (#Z159_forward.T > T#5S);   // Z159_vor
      (C)     N    "GraDB_SK".noAction
   END_STEP
   TRANSITION Z159_in_front FROM Z159_forward TO Z160_forward   // T139
      := "AlwaysFALSE";
   END_TRANSITION
   STEP Z160_forward:   // S140, max time T#10S, warning time T#7S: Step commentary / Schrittkommentar
      interlock C := "AlwaysFALSE";   // Z160_vor
      supervision V := NOT #Z160_in_front.TT AND (#Z160_forward.T > T#5S);   // Z160_vor
      (C)     N    "GraDB_SK".noAction
   END_STEP
   TRANSITION Z160_in_front FROM Z160_forward TO Z161_forward   // T140
      := "AlwaysFALSE";
   END_TRANSITION
   STEP Z161_backward:   // S41, max time T#10S, warning time T#7S: Step commentary / Schrittkommentar
      interlock C := "AlwaysFALSE";   // Z161_zur
      supervision V := NOT #Z161_back.TT AND (#Z161_backward.T > T#5S);   // Z161_zur
      (C)     N    "GraDB_SK".noAction
   END_STEP
   TRANSITION Z161_back FROM Z161_backward TO Z162_backward   // T41
      := "AlwaysFALSE";
   END_TRANSITION
   STEP Z162_backward:   // S42, max time T#10S, warning time T#7S: Step commentary / Schrittkommentar
      interlock C := "AlwaysFALSE";   // Z162_zur
      supervision V := NOT #Z162_back.TT AND (#Z162_backward.T > T#5S);   // Z162_zur
      (C)     N    "GraDB_SK".noAction
   END_STEP
   TRANSITION Z162_back FROM Z162_backward TO Z163_backward   // T42
      := "AlwaysFALSE";
   END_TRANSITION
   STEP Z163_backward:   // S43, max time T#10S, warning time T#7S: Step commentary / Schrittkommentar
      interlock C := "AlwaysFALSE";   // Z163_zur
      supervision V := NOT #Z163_back.TT AND (#Z163_backward.T > T#5S);   // Z163_zur
      (C)     N    "GraDB_SK".noAction
   END_STEP
   TRANSITION Z163_back FROM Z163_backward TO Z164_backward   // T43
      := "AlwaysFALSE";
   END_TRANSITION
   STEP Z164_backward:   // S44, max time T#10S, warning time T#7S: Step commentary / Schrittkommentar
      interlock C := "AlwaysFALSE";   // Z164_zur
      supervision V := NOT #Z164_back.TT AND (#Z164_backward.T > T#5S);   // Z164_zur
      (C)     N    "GraDB_SK".noAction
   END_STEP
   TRANSITION Z164_back FROM Z164_backward TO Z165_backward   // T44
      := "AlwaysFALSE";
   END_TRANSITION
   STEP Z165_backward:   // S45, max time T#10S, warning time T#7S: Step commentary / Schrittkommentar
      interlock C := "AlwaysFALSE";   // Z165_zur
      supervision V := NOT #Z165_back.TT AND (#Z165_backward.T > T#5S);   // Z165_zur
      (C)     N    "GraDB_SK".noAction
   END_STEP
   TRANSITION Z165_back FROM Z165_backward TO Z166_backward   // T45
      := "AlwaysFALSE";
   END_TRANSITION
   STEP Z161_forward:   // S141, max time T#10S, warning time T#7S
      interlock C := "AlwaysFALSE";   // Z161_vor
      supervision V := NOT #Z161_in_front.TT AND (#Z161_forward.T > T#5S);   // Z161_vor
      (C)     N    "GraDB_SK".noAction
   END_STEP
   TRANSITION Z161_in_front FROM Z161_forward TO Z162_forward   // T141
      := "AlwaysFALSE";
   END_TRANSITION
   STEP Z162_forward:   // S142, max time T#10S, warning time T#7S
      interlock C := "AlwaysFALSE";   // Z162_vor
      supervision V := NOT #Z162_in_front.TT AND (#Z162_forward.T > T#5S);   // Z162_vor
      (C)     N    "GraDB_SK".noAction
   END_STEP
   TRANSITION Z162_in_front FROM Z162_forward TO Z163_forward   // T142
      := "AlwaysFALSE";
   END_TRANSITION
   STEP Z163_forward:   // S143, max time T#10S, warning time T#7S
      interlock C := "AlwaysFALSE";   // Z163_vor
      supervision V := NOT #Z163_in_front.TT AND (#Z163_forward.T > T#5S);   // Z163_vor
      (C)     N    "GraDB_SK".noAction
   END_STEP
   TRANSITION Z163_in_front FROM Z163_forward TO Z164_forward   // T143
      := "AlwaysFALSE";
   END_TRANSITION
   STEP Z164_forward:   // S144, max time T#10S, warning time T#7S
      interlock C := "AlwaysFALSE";   // Z164_vor
      supervision V := NOT #Z164_in_front.TT AND (#Z164_forward.T > T#5S);   // Z164_vor
      (C)     N    "GraDB_SK".noAction
   END_STEP
   TRANSITION Z164_in_front FROM Z164_forward TO Z165_forward   // T144
      := "AlwaysFALSE";
   END_TRANSITION
   STEP Z165_forward:   // S145, max time T#10S, warning time T#7S
      interlock C := "AlwaysFALSE";   // Z165_vor
      supervision V := NOT #Z165_in_front.TT AND (#Z165_forward.T > T#5S);   // Z165_vor
      (C)     N    "GraDB_SK".noAction
   END_STEP
   TRANSITION Z165_in_front FROM Z165_forward TO Z166_forward   // T145
      := "AlwaysFALSE";
   END_TRANSITION
   STEP Z166_backward:   // S46, max time T#10S, warning time T#7S: Step commentary / Schrittkommentar
      interlock C := "AlwaysFALSE";   // Z166_zur
      supervision V := NOT #Z166_back.TT AND (#Z166_backward.T > T#5S);   // Z166_zur
      (C)     N    "GraDB_SK".noAction
   END_STEP
   TRANSITION Z166_back FROM Z166_backward TO Z167_backward   // T46
      := "AlwaysFALSE";
   END_TRANSITION
   STEP Z167_backward:   // S47, max time T#10S, warning time T#7S: Step commentary / Schrittkommentar
      interlock C := "AlwaysFALSE";   // Z167_zur
      supervision V := NOT #Z167_back.TT AND (#Z167_backward.T > T#5S);   // Z167_zur
      (C)     N    "GraDB_SK".noAction
   END_STEP
   TRANSITION Z167_back FROM Z167_backward TO Z168_backward   // T47
      := "AlwaysFALSE";
   END_TRANSITION
   STEP Z168_backward:   // S48, max time T#10S, warning time T#7S: Step commentary / Schrittkommentar
      interlock C := "AlwaysFALSE";   // Z168_zur
      supervision V := NOT #Z168_back.TT AND (#Z168_backward.T > T#5S);   // Z168_zur
      (C)     N    "GraDB_SK".noAction
   END_STEP
   TRANSITION Z168_back FROM Z168_backward TO Z169_backward   // T48
      := "AlwaysFALSE";
   END_TRANSITION
   STEP Z169_backward:   // S49, max time T#10S, warning time T#7S: Step commentary / Schrittkommentar
      interlock C := "AlwaysFALSE";   // Z169_zur
      supervision V := NOT #Z169_back.TT AND (#Z169_backward.T > T#5S);   // Z169_zur
      (C)     N    "GraDB_SK".noAction
   END_STEP
   TRANSITION Z169_back FROM Z169_backward TO Z170_backward   // T49
      := "AlwaysFALSE";
   END_TRANSITION
   STEP Z170_backward:   // S50, max time T#10S, warning time T#7S: Step commentary / Schrittkommentar
      interlock C := "AlwaysFALSE";   // Z170_zur
      supervision V := NOT #Z170_back.TT AND (#Z170_backward.T > T#5S);   // Z170_zur
      (C)     N    "GraDB_SK".noAction
   END_STEP
   TRANSITION Z170_back FROM Z170_backward TO Z171_backward   // T50
      := "AlwaysFALSE";
   END_TRANSITION
   STEP Z166_forward:   // S146, max time T#10S, warning time T#7S: Step commentary / Schrittkommentar
      interlock C := "AlwaysFALSE";   // Z166_vor
      supervision V := NOT #Z166_in_front.TT AND (#Z166_forward.T > T#5S);   // Z166_vor
      (C)     N    "GraDB_SK".noAction
   END_STEP
   TRANSITION Z166_in_front FROM Z166_forward TO Z167_forward   // T146
      := "AlwaysFALSE";
   END_TRANSITION
   STEP Z167_forward:   // S147, max time T#10S, warning time T#7S: Step commentary / Schrittkommentar
      interlock C := "AlwaysFALSE";   // Z167_vor
      supervision V := NOT #Z167_in_front.TT AND (#Z167_forward.T > T#5S);   // Z167_vor
      (C)     N    "GraDB_SK".noAction
   END_STEP
   TRANSITION Z167_in_front FROM Z167_forward TO Z168_forward   // T147
      := "AlwaysFALSE";
   END_TRANSITION
   STEP Z168_forward:   // S148, max time T#10S, warning time T#7S: Step commentary / Schrittkommentar
      interlock C := "AlwaysFALSE";   // Z168_vor
      supervision V := NOT #Z168_in_front.TT AND (#Z168_forward.T > T#5S);   // Z168_vor
      (C)     N    "GraDB_SK".noAction
   END_STEP
   TRANSITION Z168_in_front FROM Z168_forward TO Z169_forward   // T148
      := "AlwaysFALSE";
   END_TRANSITION
   STEP Z169_forward:   // S149, max time T#10S, warning time T#7S: Step commentary / Schrittkommentar
      interlock C := "AlwaysFALSE";   // Z169_vor
      supervision V := NOT #Z169_in_front.TT AND (#Z169_forward.T > T#5S);   // Z169_vor
      (C)     N    "GraDB_SK".noAction
   END_STEP
   TRANSITION Z169_in_front FROM Z169_forward TO Z170_forward   // T149
      := "AlwaysFALSE";
   END_TRANSITION
   STEP Z170_forward:   // S150, max time T#10S, warning time T#7S: Step commentary / Schrittkommentar
      interlock C := "AlwaysFALSE";   // Z170_vor
      supervision V := NOT #Z170_in_front.TT AND (#Z170_forward.T > T#5S);   // Z170_vor
      (C)     N    "GraDB_SK".noAction
   END_STEP
   TRANSITION Z170_in_front FROM Z170_forward TO Z171_forward   // T150
      := "AlwaysFALSE";
   END_TRANSITION
   STEP Z171_backward:   // S51, max time T#10S, warning time T#7S: Step commentary / Schrittkommentar
      interlock C := "AlwaysFALSE";   // Z171_zur
      supervision V := NOT #Z171_back.TT AND (#Z171_backward.T > T#5S);   // Z171_zur
      (C)     N    "GraDB_SK".noAction
   END_STEP
   TRANSITION Z171_back FROM Z171_backward TO Z172_backward   // T51
      := "AlwaysFALSE";
   END_TRANSITION
   STEP Z172_backward:   // S52, max time T#10S, warning time T#7S: Step commentary / Schrittkommentar
      interlock C := "AlwaysFALSE";   // Z172_zur
      supervision V := NOT #Z172_back.TT AND (#Z172_backward.T > T#5S);   // Z172_zur
      (C)     N    "GraDB_SK".noAction
   END_STEP
   TRANSITION Z172_back FROM Z172_backward TO Z173_backward   // T52
      := "AlwaysFALSE";
   END_TRANSITION
   STEP Z173_backward:   // S53, max time T#10S, warning time T#7S: Step commentary / Schrittkommentar
      interlock C := "AlwaysFALSE";   // Z173_zur
      supervision V := NOT #Z173_back.TT AND (#Z173_backward.T > T#5S);   // Z173_zur
      (C)     N    "GraDB_SK".noAction
   END_STEP
   TRANSITION Z173_back FROM Z173_backward TO Z174_backward   // T53
      := "AlwaysFALSE";
   END_TRANSITION
   STEP Z174_backward:   // S54, max time T#10S, warning time T#7S: Step commentary / Schrittkommentar
      interlock C := "AlwaysFALSE";   // Z174_zur
      supervision V := NOT #Z174_back.TT AND (#Z174_backward.T > T#5S);   // Z174_zur
      (C)     N    "GraDB_SK".noAction
   END_STEP
   TRANSITION Z174_back FROM Z174_backward TO Z175_backward   // T54
      := "AlwaysFALSE";
   END_TRANSITION
   STEP Z175_backward:   // S55, max time T#10S, warning time T#7S: Step commentary / Schrittkommentar
      interlock C := "AlwaysFALSE";   // Z175_zur
      supervision V := NOT #Z175_back.TT AND (#Z175_backward.T > T#5S);   // Z175_zur
      (C)     N    "GraDB_SK".noAction
   END_STEP
   TRANSITION Z175_back FROM Z175_backward TO Z176_backward   // T55
      := "AlwaysFALSE";
   END_TRANSITION
   STEP Z176_backward:   // S56, max time T#10S, warning time T#7S: Step commentary / Schrittkommentar
      interlock C := "AlwaysFALSE";   // Z176_zur
      supervision V := NOT #Z176_back.TT AND (#Z176_backward.T > T#5S);   // Z176_zur
      (C)     N    "GraDB_SK".noAction
   END_STEP
   TRANSITION Z176_back FROM Z176_backward TO Z177_backward   // T56
      := "AlwaysFALSE";
   END_TRANSITION
   STEP Z177_backward:   // S57, max time T#10S, warning time T#7S: Step commentary / Schrittkommentar
      interlock C := "AlwaysFALSE";   // Z177_zur
      supervision V := NOT #Z177_back.TT AND (#Z177_backward.T > T#5S);   // Z177_zur
      (C)     N    "GraDB_SK".noAction
   END_STEP
   TRANSITION Z177_back FROM Z177_backward TO Z178_backward   // T57
      := "AlwaysFALSE";
   END_TRANSITION
   STEP Z178_backward:   // S58, max time T#10S, warning time T#7S: Step commentary / Schrittkommentar
      interlock C := "AlwaysFALSE";   // Z178_zur
      supervision V := NOT #Z178_back.TT AND (#Z178_backward.T > T#5S);   // Z178_zur
      (C)     N    "GraDB_SK".noAction
   END_STEP
   TRANSITION Z178_back FROM Z178_backward TO Z179_backward   // T58
      := "AlwaysFALSE";
   END_TRANSITION
   STEP Z179_backward:   // S59, max time T#10S, warning time T#7S: Step commentary / Schrittkommentar
      interlock C := "AlwaysFALSE";   // Z179_zur
      supervision V := NOT #Z179_back.TT AND (#Z179_backward.T > T#5S);   // Z179_zur
      (C)     N    "GraDB_SK".noAction
   END_STEP
   TRANSITION Z179_back FROM Z179_backward TO Z180_backward   // T59
      := "AlwaysFALSE";
   END_TRANSITION
   STEP Z180_backward:   // S60, max time T#10S, warning time T#7S: Step commentary / Schrittkommentar
      interlock C := "AlwaysFALSE";   // Z180_zur
      supervision V := NOT #Z180_back.TT AND (#Z180_backward.T > T#5S);   // Z180_zur
      (C)     N    "GraDB_SK".noAction
   END_STEP
   TRANSITION Z180_back FROM Z180_backward TO END   // T60
      := "AlwaysFALSE";
   END_TRANSITION
   STEP Z171_forward:   // S151, max time T#10S, warning time T#7S
      interlock C := "AlwaysFALSE";   // Z171_vor
      supervision V := NOT #Z171_in_front.TT AND (#Z171_forward.T > T#5S);   // Z171_vor
      (C)     N    "GraDB_SK".noAction
   END_STEP
   TRANSITION Z171_in_front FROM Z171_forward TO Z172_forward   // T151
      := "AlwaysFALSE";
   END_TRANSITION
   STEP Z172_forward:   // S152, max time T#10S, warning time T#7S
      interlock C := "AlwaysFALSE";   // Z172_vor
      supervision V := NOT #Z172_in_front.TT AND (#Z172_forward.T > T#5S);   // Z172_vor
      (C)     N    "GraDB_SK".noAction
   END_STEP
   TRANSITION Z172_in_front FROM Z172_forward TO Z173_forward   // T152
      := "AlwaysFALSE";
   END_TRANSITION
   STEP Z173_forward:   // S153, max time T#10S, warning time T#7S
      interlock C := "AlwaysFALSE";   // Z173_vor
      supervision V := NOT #Z173_in_front.TT AND (#Z173_forward.T > T#5S);   // Z173_vor
      (C)     N    "GraDB_SK".noAction
   END_STEP
   TRANSITION Z173_in_front FROM Z173_forward TO Z174_forward   // T153
      := "AlwaysFALSE";
   END_TRANSITION
   STEP Z174_forward:   // S154, max time T#10S, warning time T#7S
      interlock C := "AlwaysFALSE";   // Z174_vor
      supervision V := NOT #Z174_in_front.TT AND (#Z174_forward.T > T#5S);   // Z174_vor
      (C)     N    "GraDB_SK".noAction
   END_STEP
   TRANSITION Z174_in_front FROM Z174_forward TO Z175_forward   // T154
      := "AlwaysFALSE";
   END_TRANSITION
   STEP Z175_forward:   // S155, max time T#10S, warning time T#7S
      interlock C := "AlwaysFALSE";   // Z175_vor
      supervision V := NOT #Z175_in_front.TT AND (#Z175_forward.T > T#5S);   // Z175_vor
      (C)     N    "GraDB_SK".noAction
   END_STEP
   TRANSITION Z175_in_front FROM Z175_forward TO Z176_forward   // T155
      := "AlwaysFALSE";
   END_TRANSITION
   STEP Z176_forward:   // S156, max time T#10S, warning time T#7S: Step commentary / Schrittkommentar
      interlock C := "AlwaysFALSE";   // Z176_vor
      supervision V := NOT #Z176_in_front.TT AND (#Z176_forward.T > T#5S);   // Z176_vor
      (C)     N    "GraDB_SK".noAction
   END_STEP
   TRANSITION Z176_in_front FROM Z176_forward TO Z177_forward   // T156
      := "AlwaysFALSE";
   END_TRANSITION
   STEP Z177_forward:   // S157, max time T#10S, warning time T#7S: Step commentary / Schrittkommentar
      interlock C := "AlwaysFALSE";   // Z177_vor
      supervision V := NOT #Z177_in_front.TT AND (#Z177_forward.T > T#5S);   // Z177_vor
      (C)     N    "GraDB_SK".noAction
   END_STEP
   TRANSITION Z177_in_front FROM Z177_forward TO Z178_forward   // T157
      := "AlwaysFALSE";
   END_TRANSITION
   STEP Z178_forward:   // S158, max time T#10S, warning time T#7S: Step commentary / Schrittkommentar
      interlock C := "AlwaysFALSE";   // Z178_vor
      supervision V := NOT #Z178_in_front.TT AND (#Z178_forward.T > T#5S);   // Z178_vor
      (C)     N    "GraDB_SK".noAction
   END_STEP
   TRANSITION Z178_in_front FROM Z178_forward TO Z179_forward   // T158
      := "AlwaysFALSE";
   END_TRANSITION
   STEP Z179_forward:   // S159, max time T#10S, warning time T#7S: Step commentary / Schrittkommentar
      interlock C := "AlwaysFALSE";   // Z179_vor
      supervision V := NOT #Z179_in_front.TT AND (#Z179_forward.T > T#5S);   // Z179_vor
      (C)     N    "GraDB_SK".noAction
   END_STEP
   TRANSITION Z179_in_front FROM Z179_forward TO Z180_forward   // T159
      := "AlwaysFALSE";
   END_TRANSITION
   STEP Z180_forward:   // S160, max time T#10S, warning time T#7S: Step commentary / Schrittkommentar
      interlock C := "AlwaysFALSE";   // Z180_vor
      supervision V := NOT #Z180_in_front.TT AND (#Z180_forward.T > T#5S);   // Z180_vor
      (C)     N    "GraDB_SK".noAction
   END_STEP
   TRANSITION Z180_in_front FROM Z180_forward TO END   // T160
      := "AlwaysFALSE";
   END_TRANSITION

   // permanent post-instructions
   NETWORK 1
   TITLE = HMI Lite Pass on data / HMI Lite Daten weiterreichen
      "LTLL_ManualGraphInterlock"(ManualGraphExtOutput := #extBlock.output,
                              ManualGraphControlScreen := "LTLL_ManualGraphControl_OP70".screen[0]);
   NETWORK 2
   TITLE = Report step error / Schrittkettenfehler melden
      "SysFC_NumOfSQErrors"(FLT := #RT_DATA.SQ_FLAGS.ERR_FLT,
                            Fault_SQ := "AnwDB_OperatingModes_OP70".BA[0].error_report_SK,
                            NumOf_Fault_SQ := "AnwDB_ZP_Alarm_OP70".FaultsNoSK_ST1);
END_FUNCTION_BLOCK
